(* Logix 5000 project; controller Proyecto_Lavadora Emulate 5570 rev 33.11; software revision 33.00 *)

TASK T00_MainTask (continuous, watchdog 500 ms) : P00_MainProgram

MODULES
   Local : Emulate 5570 (ICP 2, rev 33.11)
END_MODULES

VAR_GLOBAL   (* controller tags *)
   I00_S_Cerrado : BOOL := 1;
   I01_S_Abierto : BOOL;
   I02_B_Arranque : BOOL;
   I03_B_Apagado : BOOL;
   O00_P_Lavado_Enjuague : BOOL;
   O01_P_Centrifugado : BOOL;
   O02_Seguros_Puertas : BOOL;
   O03_P_Llenado : BOOL;
   O04_P_Vaciado : BOOL;
   T00_Llenado : TIMER := (PRE := 5000);
   T01_Vaciado : TIMER := (PRE := 5000);
   T02_Lavado : TIMER := (PRE := 12000);
   T03_Enjuague : TIMER := (PRE := 8000);
   T04_Centrifugado : TIMER := (PRE := 10000);
   T05_Frenos : TIMER := (PRE := 3000);
END_VAR

PROGRAM P00_MainProgram   (* main routine R00_MainRoutine *)

ROUTINE R00_MainRoutine   (* ladder *)
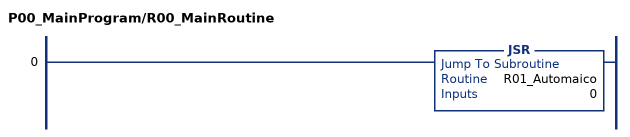
   0: JSR(R01_Automaico,0);
END_ROUTINE

ROUTINE R01_Automaico   (* ladder *)
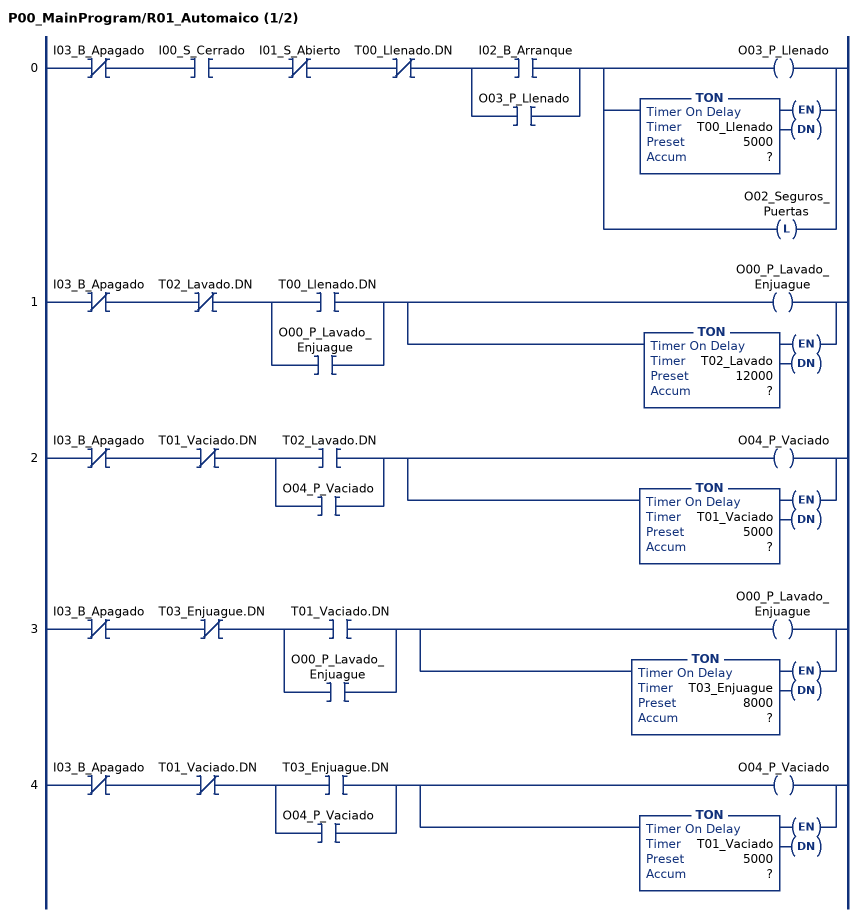
   0: XIO(I03_B_Apagado)XIC(I00_S_Cerrado)XIO(I01_S_Abierto)XIO(T00_Llenado.DN)[XIC(I02_B_Arranque) ,XIC(O03_P_Llenado) ][OTE(O03_P_Llenado) ,TON(T00_Llenado,?,?) ,OTL(O02_Seguros_Puertas) ];
   1: XIO(I03_B_Apagado)XIO(T02_Lavado.DN)[XIC(T00_Llenado.DN) ,XIC(O00_P_Lavado_Enjuague) ][OTE(O00_P_Lavado_Enjuague) ,TON(T02_Lavado,?,?) ];
   2: XIO(I03_B_Apagado)XIO(T01_Vaciado.DN)[XIC(T02_Lavado.DN) ,XIC(O04_P_Vaciado) ][OTE(O04_P_Vaciado) ,TON(T01_Vaciado,?,?) ];
   3: XIO(I03_B_Apagado)XIO(T03_Enjuague.DN)[XIC(T01_Vaciado.DN) ,XIC(O00_P_Lavado_Enjuague) ][OTE(O00_P_Lavado_Enjuague) ,TON(T03_Enjuague,?,?) ];
   4: XIO(I03_B_Apagado)XIO(T01_Vaciado.DN)[XIC(T03_Enjuague.DN) ,XIC(O04_P_Vaciado) ][OTE(O04_P_Vaciado) ,TON(T01_Vaciado,?,?) ];
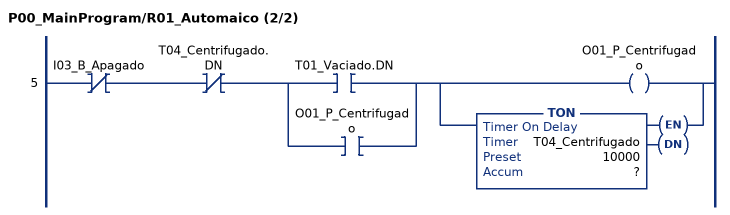
   5: XIO(I03_B_Apagado)XIO(T04_Centrifugado.DN)[XIC(T01_Vaciado.DN) ,XIC(O01_P_Centrifugado) ][OTE(O01_P_Centrifugado) ,TON(T04_Centrifugado,?,?) ];
END_ROUTINE
END_PROGRAM
